FUNCTION_BLOCK MulticastConveyorCTL (* Basic Function Block Type *)
  (* Standard: 61499-2 *)
  (* Version 0.2, 2003-12-04, JHC, Rockwell Automation, Renamed for better indexing. *)
  (* Version 0.1, 2002-11-05, JHC, Rockwell Automation, Corrected missing ST element in Algorithm REQ. *)
  (* Version 0.0, 2000-05-30, JHC, Rockwell Automation *)
  (* Compiler header: package fb.rt.cs725.T17; *)
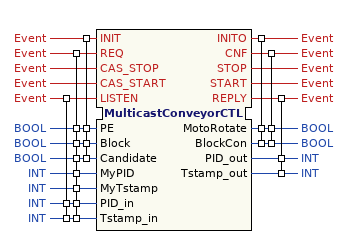
  EVENT_INPUT
    INIT WITH PE, Block, Candidate; (* Initialization Request *)
    REQ WITH PE, Block, Candidate, MyPID, MyTstamp, PID_in, Tstamp_in; (* Normal Execution Request *)
    CAS_STOP;
    CAS_START;
    LISTEN WITH PID_in, Tstamp_in;
  END_EVENT
  EVENT_OUTPUT
    INITO WITH MotoRotate, BlockCon; (* Initialization Confirm *)
    CNF WITH MotoRotate, BlockCon; (* Execution Confirmation *)
    STOP;
    START;
    REPLY WITH PID_out, Tstamp_out;
  END_EVENT
  VAR_INPUT
    PE : BOOL; (* Input event qualifier *)
    Block : BOOL;
    Candidate : BOOL;
    MyPID : INT;
    MyTstamp : INT;
    PID_in : INT;
    Tstamp_in : INT;
  END_VAR
  VAR_OUTPUT
    MotoRotate : BOOL; (* Output event qualifier *)
    BlockCon : BOOL;
    PID_out : INT;
    Tstamp_out : INT;
  END_VAR
  VAR
    lastPE : BOOL := 1;
    lastBlock : BOOL := 0;
    MeFirst : BOOL;
    YouFirst : BOOL;
    LampClock : UINT;
  END_VAR
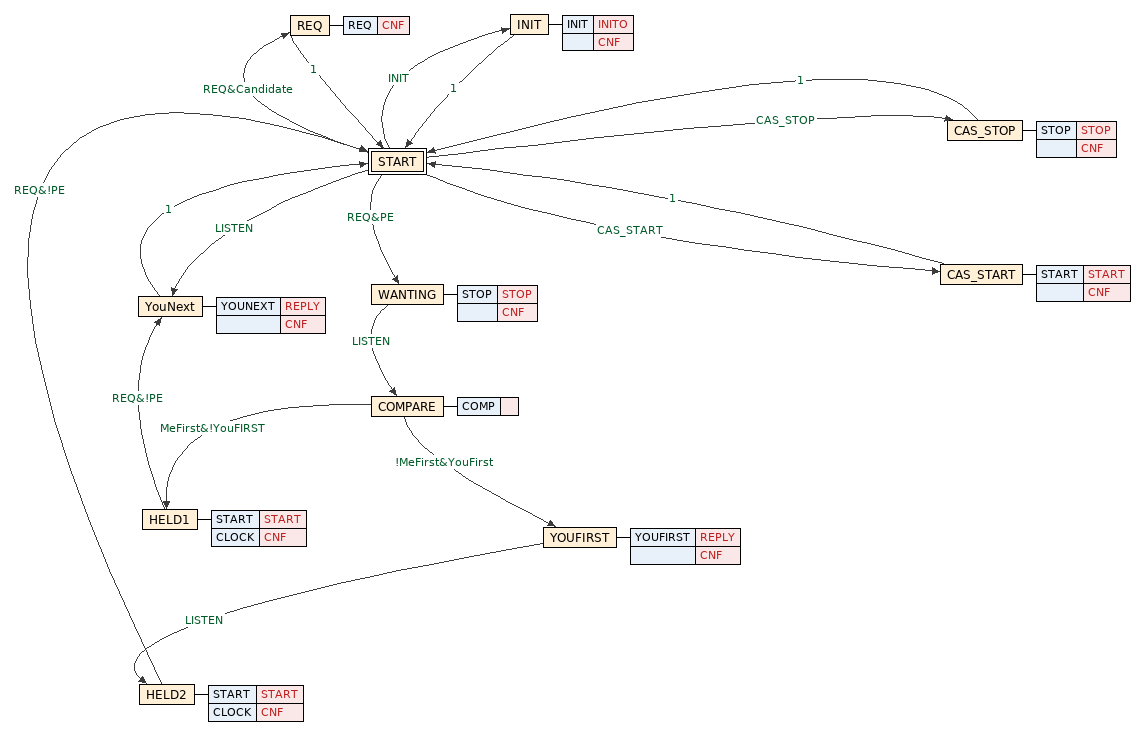
  EC_STATES
    START; (* Initial State *)
    INIT : INIT -> INITO, -> CNF; (* Initialization *)
    REQ : REQ -> CNF; (* Normal execution *)
    CAS_START : START -> START, -> CNF;
    CAS_STOP : STOP -> STOP, -> CNF;
    WANTING : STOP -> STOP, -> CNF;
    COMPARE : COMP;
    HELD1 : START -> START, CLOCK -> CNF;
    HELD2 : START -> START, CLOCK -> CNF;
    YOUFIRST : YOUFIRST -> REPLY, -> CNF;
    YouNext : YOUNEXT -> REPLY, -> CNF;
  END_STATES
  EC_TRANSITIONS
    START TO INIT := INIT;
    INIT TO START := 1;
    START TO REQ := REQ&Candidate;
    REQ TO START := 1;
    START TO CAS_START := CAS_START;
    CAS_START TO START := 1;
    START TO CAS_STOP := CAS_STOP;
    CAS_STOP TO START := 1;
    START TO WANTING := REQ&PE;
    WANTING TO COMPARE := LISTEN;
    YOUFIRST TO HELD2 := LISTEN;
    COMPARE TO YOUFIRST := !MeFirst&YouFirst;
    COMPARE TO HELD1 := MeFirst&!YouFIRST;
    HELD1 TO YouNext := REQ&!PE;
    HELD2 TO START := REQ&!PE;
    YouNext TO START := 1;
    START TO YouNext := LISTEN;
  END_TRANSITIONS
  ALGORITHM INIT IN ST: (* Initialization algorithm *)
MotoRotate := TRUE;
Block := FALSE;
LampClock := MyTstamp;
MeFirst := false;
Youfirst := false;

System.out.println(this + " " + MotoRotate);
System.out.println(MotoRotate);
  END_ALGORITHM
  ALGORITHM REQ IN Java: (* Normally executed algorithm *)
System.out.println("In REQ State");

MeFirst.value = false;
Youfirst.value = false;

if(lastPE.value!=PE.value){
if(!PE.value){
BlockCon.value=true;
System.out.println("BlockCon = true");
}
else{
BlockCon.value=false;
System.out.println("BlockCon = false");
}
lastPE.value=PE.value;
}
if(lastBlock.value!=Block.value){
if(Block.value){
STOP.serviceEvent(this);
MotoRotate.value=false;
System.out.println("Cas Stop");
}
else{
START.serviceEvent(this);
MotoRotate.value=true;
System.out.println("Cas Start");
}
lastBlock.value=Block.value;
}

LampClock.value++;
  END_ALGORITHM
  ALGORITHM START IN ST:
MotoRotate:=TRUE;
System.out.println(this + " Start " + MotoRotate);
  END_ALGORITHM
  ALGORITHM STOP IN ST:
MotoRotate := FALSE;
System.out.println(this + " Stop " + MotoRotate);
  END_ALGORITHM
  ALGORITHM COMP IN Java:
if(MyTstamp>Tstamp_in)|(MyPID<PID_in){
MeFirst.value = true;
Youfirst.value = false;
} elseif (MyTstamp<Tstamp_in)|(MyPID>PID_in){
MeFirst.value = false;
Youfirst.value = true;
}
  END_ALGORITHM
  ALGORITHM YOUFIRST IN Java:
System.out.println("Clock is: " + LampClock.valu);
System.out.println("ID is: " + MyPID.value);

Tstamp_out.value = LampClock.value;
PID_out.value = MyPID.value;
  END_ALGORITHM
  ALGORITHM CLOCK IN Java:
LampClock.value = Tstamp_in.value;
  END_ALGORITHM
  ALGORITHM YOUNEXT IN Java:
Tstamp_out.value = LampClock.value;
PID_out.value = MyPID.value;
  END_ALGORITHM
END_FUNCTION_BLOCK
